// TIA Portal V20 export
DATA_BLOCK "control"   // DB6
{ S7_Optimized_Access := 'TRUE' }
// stored: InstanceOfName UDT_control, InstanceOfType UDT
"UDT_control"
   // VAR
   //    resetCounters { ExternalVisible := 'False'} : DInt;
   //    startTaktTimeCnt { ExternalVisible := 'False'} : DInt;
   //    stopTaktTimeCnt { ExternalVisible := 'False'} : DInt;
   //    actualMinus1 : DInt;
   //    actualPlus1 : DInt;
   //    okMinus1 : DInt;
   //    okPlus1 : DInt;
   // END_VAR
BEGIN
END_DATA_BLOCK
